// TIA Portal V20 export
TYPE "CMInterface"
   STRUCT
      CM_DI001 { ExternalAccessible := 'False'; ExternalVisible := 'False'; ExternalWritable := 'False'} : "CMInterface_DI";
      CM_DO001 { ExternalAccessible := 'False'; ExternalVisible := 'False'; ExternalWritable := 'False'} : "CMInterface_DO";
      CM_AI001 { ExternalAccessible := 'False'; ExternalVisible := 'False'; ExternalWritable := 'False'} : "CMInterface_AI";
      CM_AO001 { ExternalAccessible := 'False'; ExternalVisible := 'False'; ExternalWritable := 'False'} : "CMInterface_AO";
      CM_VSD001 { ExternalAccessible := 'False'; ExternalVisible := 'False'; ExternalWritable := 'False'} : "CMInterface_VSD";
      CM_MOT001 { ExternalAccessible := 'False'; ExternalVisible := 'False'; ExternalWritable := 'False'} : "CMInterface_MOT";
      CM_VLV001 { ExternalAccessible := 'False'; ExternalVisible := 'False'; ExternalWritable := 'False'} : "CMInterface_VLV";
      CM_CONTVLV001 { ExternalAccessible := 'False'; ExternalVisible := 'False'; ExternalWritable := 'False'} : "CMInterface_CONTVLV";
   END_STRUCT;
END_TYPE
